// TwinCAT 3 PLC project AdventOfCode2024_Day02
// ProgramVersion: 3.1.4026.12
// libraries:
//   SH_FileReader, * (Stefan Halder)
//   Tc2_Standard, * (Beckhoff Automation GmbH)
//   Tc2_System, * (Beckhoff Automation GmbH)
// project tree:
//   DUTs/ ERROR.TcDUT
//   GVLs/ GLOBAL_CONSTANTS.TcGVL
//   / PlcTask.TcTTO
//   POUs/FileReader/DUTs/ STATE.TcDUT (not stored)
//   POUs/FileReader/ FileReader.TcPOU
//   POUs/ MAIN.TcPOU
// real-time tasks:
//   TASK PlcTask: cycle T#10ms, priority 20, ADS port 350

CONFIGURATION AdventOfCode2024_Day02
    RESOURCE PLC ON TwinCAT3
        TASK PlcTask(INTERVAL := T#10ms, PRIORITY := 20);
        PROGRAM MAIN WITH PlcTask : MAIN;
    END_RESOURCE
END_CONFIGURATION

// ---- DUTs/ERROR.TcDUT
TYPE ERROR :
STRUCT
	bError : BOOL;
	nErrorCode : UDINT;
	dtCurrentTime : DT;
END_STRUCT
END_TYPE

// ---- GVLs/GLOBAL_CONSTANTS.TcGVL
VAR_GLOBAL CONSTANT
	iC_MAX_NUM_LINES_IN_FILE : UINT := 1000;
	iC_MAX_STRING_LENGTH : UINT := 25;
END_VAR

// ---- POUs/MAIN.TcPOU
PROGRAM MAIN
VAR
	sFilePath : T_MaxString := 'E:\Projects\Twincat\AdventOfCode\Day02\Day2Input.txt'; //'C:\temp\HelloWorld.txt';// 
	fb_FileReader : SH_FileReader.FileReader;
	bFileReaderDone : BOOL;	
		
	stFileReaderError : SH_FileReader.ERROR;

	fb_Analysis : Analysis;
	
	bReadFile : BOOL;
	bAnalyzeFile : BOOL;
END_VAR

fb_FileReader();

bFileReaderDone := fb_FileReader.ReadFile(bExecute := bReadFile, sFilePath := sFilePath, stError => stFileReaderError);
IF bReadFile THEN
	bReadFile := FALSE;
END_IF

IF bAnalyzeFile THEN
	bAnalyzeFile := FALSE;
	FOR iLoopIndexFileContentArray := 0 TO iC_MAX_NUM_LINES_IN_FILE-1 DO
		sTempString := fb_FileReader.GetLineByIndex(iLoopIndexFileContentArray);
		nNumElementsInLine := ((LEN(sTempString) + 1)/3)-1;
		FOR iLoopIndexString := 0 TO nNumElementsInLine DO
			arsStringArray[iLoopIndexString] := MID(sTempString, 2, iLoopIndexString*3+1);
			arnNumberArray[iLoopIndexString] := TO_UINT(arsStringArray[iLoopIndexString]);
		END_FOR
		bIncreasing := THIS^.CheckIncreasing();
	END_FOR
END_IF

METHOD CheckIncreasing : BOOL
VAR
	iLoopIndex : UINT;
	bStepIncreasing : BOOL;
	bIncreasing : BOOL;
END_VAR
bIncreasing := TRUE;
FOR iLoopIndex := 0 TO nNumElementsInLine DO
	bStepIncreasing := arnNumberArray[iLoopIndex] < arnNumberArray[iLoopIndex+1];
	bIncreasing := bIncreasing AND bStepIncreasing;			
END_FOR
CheckIncreasing := bIncreasing;
END_METHOD

END_PROGRAM

// ---- POUs/FileReader/FileReader.TcPOU
FUNCTION_BLOCK FileReader
VAR
	_bBusy : BOOL;
	_sFilePath : STRING;
	_arsFileContent : ARRAY [0..iC_MAX_NUM_LINES_IN_FILE] OF STRING(iC_MAX_STRING_LENGTH);
	
	fbi_FileOpen : FB_FileOpen;
	fbi_FileGets : FB_FileGets;
	fbi_FileClose : FB_FileClose;
	
	eState : STATE := STATE.Idle;
	
	hFileHandle : UINT;
	iFileContentNextIndex : UINT;
	stError : ERROR;
END_VAR

CASE eState OF
	State.Idle:
		// Do nothing
	State.OpenFile:
		_bBusy := TRUE;
		iFileContentNextIndex := 0;
		MEMSET(ADR(_arsFileContent), 0, SIZEOF(_arsFileContent));
		fbi_FileOpen(sPathName := sFilePath, nMode := FOPEN_MODEREAD OR FOPEN_MODETEXT, ePath := PATH_GENERIC, bExecute := TRUE, bError => stError.bError, nErrId => stError.nErrorCode);
		eState := STATE.OpenFileAwaitFinish;
		
	State.OpenFileAwaitFinish:
		fbi_FileOpen(bExecute := FALSE, hFile => hFileHandle, bError => stError.bError, nErrId => stError.nErrorCode);
		IF NOT fbi_FileOpen.bBusy THEN
			IF NOT stError.bError THEN
				eState := STATE.ReadFile;
			ELSE
				eState := STATE.Error;
			END_IF
		END_IF
		
	State.ReadFile:
		fbi_FileGets(hFile := hFileHandle, bExecute := TRUE, bError => stError.bError, nErrId => stError.nErrorCode);
		eState := STATE.ReadFileAwaitFinish;
		
	State.ReadFileAwaitFinish:
		fbi_FileGets(bExecute := FALSE, bError => stError.bError, nErrId => stError.nErrorCode);
		IF NOT fbi_FileGets.bBusy THEN
			IF NOT stError.bError THEN
				_arsFileContent[iFileContentNextIndex] := fbi_FileGets.sLine;
				IF fbi_FileGets.bEOF THEN
					eState := STATE.CloseFile;
				ELSE
					eState := STATE.ReadFile;
					iFileContentNextIndex := iFileContentNextIndex+1;	
				END_IF
			ELSE
				eState := STATE.Error;
			END_IF	
		END_IF
		
	State.CloseFile:
		fbi_FileClose(hFile := hFileHandle, bExecute := TRUE, bError => stError.bError, nErrId => stError.nErrorCode);
		eState := STATE.CloseFileAwaitFinish;
		
	State.CloseFileAwaitFinish:
		fbi_FileClose(bExecute := FALSE, bError => stError.bError, nErrId => stError.nErrorCode);
		IF NOT fbi_FileClose.bBusy THEN
			IF NOT stError.bError THEN
				eState := STATE.Idle;
			ELSE
				eState := STATE.Error;
			END_IF
			_bBusy := FALSE;
			hFileHandle := 0;
		END_IF
		
	State.Error:
		eState := STATE.Idle;
END_CASE

PROPERTY arsFileContent : ARRAY [0..iC_MAX_NUM_LINES_IN_FILE] OF STRING(iC_MAX_STRING_LENGTH)
GET
arsFileContent := _arsFileContent;
END_GET
END_PROPERTY

PROPERTY bBusy : BOOL
GET
bBusy := _bBusy;
END_GET
END_PROPERTY

METHOD GetLineByIndex : STRING
VAR_INPUT
	iIndex : UINT;
END_VAR
GetLineByIndex := _arsFileContent[iIndex];
END_METHOD

METHOD ReadFile : BOOL
VAR_INPUT
	sFilePath : STRING;
END_VAR
_bBusy := TRUE;
_sFilePath := sFilePath;
IF eState = STATE.Idle THEN
	eState := STATE.OpenFile;
END_IF
ReadFile := NOT _bBusy AND NOT stError.bError;
END_METHOD

PROPERTY sFilePath : STRING
GET
sFilePath := _sFilePath;
END_GET
SET
_sFilePath := sFilePath;
END_SET
END_PROPERTY

END_FUNCTION_BLOCK
